// TIA Portal V16 export
// export: Created 2025-05-30T16:30:31.9185672Z, ExportSetting WithDefaults, DisplayName Totally Integrated Automation Portal, DisplayVersion V16, DisplayName TIA Portal Version Control Interface, DisplayVersion V16, DisplayName TIA Portal Openness, DisplayVersion V16, DisplayName STEP 7 Professional, DisplayVersion V16, DisplayName STEP 7 Safety, DisplayVersion V16, DisplayName WinCC Advanced, DisplayVersion V16
DATA_BLOCK "FB_EncoderFeedback_Aanvoerband"   // DB78
VERSION : 0.1
// stored: AutoNumber true, InstanceOfName FB_EncoderFeedback_Degree, InstanceOfType FB
"FB_EncoderFeedback_Degree"
   // VAR_INPUT
   //    CounterTag { ExternalVisible := 'False'; ExternalWritable := 'False'} : Int;
   //    Position_Offset { ExternalVisible := 'False'; ExternalWritable := 'False'} : Real;
   //    Pulsfactor { ExternalVisible := 'False'; ExternalWritable := 'False'} : Real;
   //    Position_Correction { ExternalVisible := 'False'; ExternalWritable := 'False'} : Real;
   //    ReferenceRun_Command { ExternalVisible := 'False'; ExternalWritable := 'False'} : Bool;
   //    ReferenceSwitch { ExternalVisible := 'False'; ExternalWritable := 'False'} : Bool;
   //    ReferencePosition { ExternalVisible := 'False'; ExternalWritable := 'False'} : Int;
   // END_VAR
   // VAR_OUTPUT
   //    Scaled_Position { ExternalVisible := 'False'; ExternalWritable := 'False'} : Real;
   //    Actual_Enc_Pos { ExternalVisible := 'False'; ExternalWritable := 'False'} : Real;
   //    AxisDB_Connection { ExternalVisible := 'False'; ExternalWritable := 'False'} : Real;
   // END_VAR
BEGIN
END_DATA_BLOCK
